Staubli VAL3: listdel.pgx

public program listdel(num x_nIndex (dimensions=1))
  local num l_nSize
begin
  //
  // Staubli Copyright 2005 toneage
  //
  l_nSize=size(sItems)-1
  if ((x_nIndex>=0) and (x_nIndex<=l_nSize))
    if l_nSize>0
      delete(sItems[x_nIndex])
      delete(bReadWrite[x_nIndex])
    else
      sItems=""
      bReadWrite=true
    endIf
  endIf
end
